Universal Robots PolyScope program: vino 4binf.urp

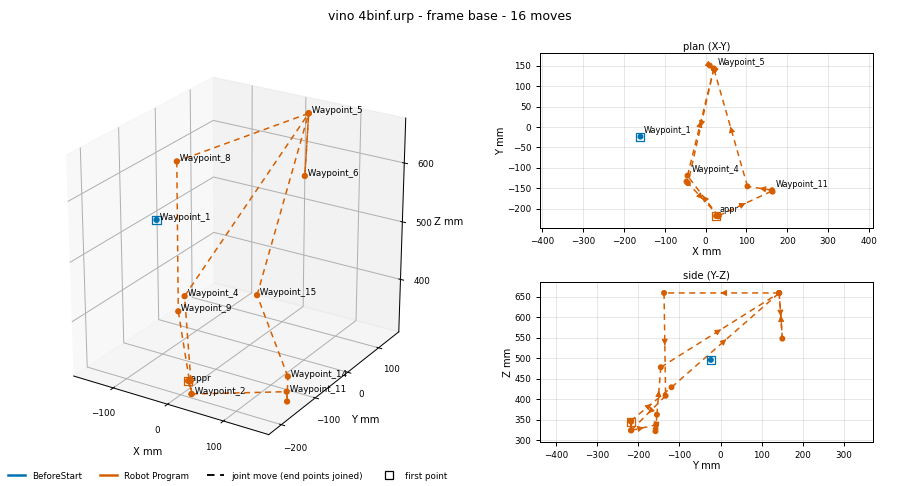
[picture p0: tool path of vino 4binf.urp in frame base, 16 of 16 moves have a stored position in this frame; points joined in program order, loops and branches not executed]
Program vino 4binf (installation=default directory=/programs createdIn=3.15.8.106339 lastSavedIn=3.15.8.106339 robotSerialNumber=2023330215)
Calibrated DH parameters: a=[-0.000158, -0.243568, -0.211872, 0.000029, -0.000046, 0]; d=[0.151957, 0.552568, 8.396945, -8.837237, 0.085345, 0.082393]; alpha=[1.571201, -0.003022, 0.002719, 1.570411, -1.571935, 0]; deltaTheta=[0.000034, -0.006936, 0.121129, -0.114397, -0.000018, 0.00002]
BeforeStart
  MoveJ speed 60 deg/s, acceleration 80 deg/s^2 (useActiveTCP=true)
    Waypoint Waypoint_1: TCP in base x=-159.567 y=-23.557 z=496.076 mm, rx=0.0292 ry=0.0156 rz=0.8759 rad; joints [-35.648, -8.811, -153.056, 70.106, 89.674, 175.859] deg; flange x=-163.543 y=-20.575 z=341.155 mm, rx=0.0292 ry=0.0156 rz=0.8759 rad
    URCap SG Grip (OnRobot, OnRobot A/S) dataModel(sg-target-width-percent=86.0)
Robot Program (runOnlyOnce=false)
  var_1 :=  (valueSource=Operator message=vino rosso:1, vino bianco:2 valueType=Integer)
  If var_1==1
    MoveJ speed 60 deg/s, acceleration 80 deg/s^2 (useActiveTCP=true)
      Waypoint appr: TCP in base x=25.587 y=-217.557 z=345.361 mm, rx=2.1967 ry=1.4969 rz=-0.0064 rad; joints [-47.133, -54.408, -74.542, -113.583, 85.897, 153.346] deg; flange x=-14.398 y=-157.633 z=482.603 mm, rx=2.1967 ry=1.4969 rz=-0.0064 rad
      Waypoint Waypoint_2: TCP in base x=31.419 y=-217.434 z=324.644 mm, rx=2.246 ry=1.4994 rz=0.0175 rad; joints [-47.147, -53.734, -79.907, -111.195, 86.968, 154.753] deg; flange x=-6.909 y=-163.472 z=464.801 mm, rx=2.246 ry=1.4994 rz=0.0175 rad
      URCap SG Grip (OnRobot, OnRobot A/S) dataModel(sg-target-width-percent=20.0, payload-weight=2.0)
      Waypoint Waypoint_3: TCP in base x=31.206 y=-218.665 z=347.338 mm, rx=2.2913 ry=1.5328 rz=-0.0001 rad; joints [-47.151, -61.647, -65.94, -120.54, 86.724, 154.677] deg; flange x=-1.134 y=-170.293 z=491.002 mm, rx=2.2913 ry=1.5328 rz=-0.0001 rad
      Waypoint Waypoint_4: TCP in base x=-44.405 y=-119.172 z=429.403 mm, rx=1.9047 ry=1.2932 rz=0.1456 rad; joints [-47.179, -40.473, -51.871, -129.238, 89.687, 154.311] deg; flange x=-122.306 y=-33.483 z=532.426 mm, rx=1.9047 ry=1.2932 rz=0.1456 rad
      MoveJ speed 60 deg/s, acceleration 80 deg/s^2 (useActiveTCP=true)
        Waypoint Waypoint_5: TCP in base x=20.05 y=142.744 z=658.935 mm, rx=1.2454 ry=-1.634 rz=-1.9818 rad; joints [-217.962, -70.658, 4.281, -114.39, 87.004, 154.418] deg; flange x=137.145 y=41.214 z=661.225 mm, rx=1.2454 ry=-1.634 rz=-1.9818 rad
        Wait Sleep waitTime=2
        Waypoint Waypoint_6: TCP in base x=9.998 y=150.468 z=547.731 mm, rx=1.5437 ry=-1.9858 rz=-1.5274 rad; joints [-217.959, -70.753, 4.268, -140.009, 87.003, 154.445] deg; flange x=114.246 y=59.022 z=616.978 mm, rx=1.5437 ry=-1.9858 rz=-1.5274 rad
        Wait Sleep waitTime=1
        Waypoint Waypoint_7: TCP in base x=20.075 y=142.736 z=658.923 mm, rx=1.2454 ry=-1.634 rz=-1.9819 rad; joints [-217.962, -70.654, 4.28, -114.394, 87.002, 154.414] deg; flange x=137.166 y=41.2 z=661.214 mm, rx=1.2454 ry=-1.634 rz=-1.9819 rad
        MoveJ speed 60 deg/s, acceleration 80 deg/s^2 (useActiveTCP=true)
          Waypoint Waypoint_8: TCP in base x=-43.492 y=-137.422 z=658.955 mm, rx=1.3394 ry=0.8543 rz=0.1901 rad; joints [-47.527, -70.659, 4.283, -114.386, 87.005, 154.417] deg; flange x=-142.09 y=-17.846 z=661.232 mm, rx=1.3394 ry=0.8543 rz=0.1901 rad
          Waypoint Waypoint_9: TCP in base x=-46.796 y=-133.623 z=408.73 mm, rx=1.9227 ry=1.2652 rz=0.0928 rad; joints [-47.145, -35.139, -63.529, -123.112, 86.887, 154.749] deg; flange x=-118.779 y=-43.172 z=511.988 mm, rx=1.9227 ry=1.2652 rz=0.0928 rad
          Waypoint Waypoint_10: TCP in base x=31.441 y=-217.42 z=324.618 mm, rx=2.246 ry=1.4996 rz=0.0176 rad; joints [-47.142, -53.734, -79.911, -111.196, 86.97, 154.751] deg; flange x=-6.888 y=-163.473 z=464.781 mm, rx=2.246 ry=1.4996 rz=0.0176 rad
          URCap SG Release (OnRobot, OnRobot A/S) dataModel(sg-target-width-percent=80.0)
  ElseIf var_1==2
    MoveJ speed 60 deg/s, acceleration 80 deg/s^2 (useActiveTCP=true)
      Waypoint Waypoint_11: TCP in base x=161.964 y=-156.646 z=337.88 mm, rx=1.2717 ry=2.6052 rz=-0.07 rad; joints [-4.628, -69.227, -57.746, -130.989, 82.548, 136.638] deg; flange x=131.859 y=-133.75 z=488.195 mm, rx=1.2717 ry=2.6052 rz=-0.07 rad
      Waypoint Waypoint_12: TCP in base x=163.817 y=-158.291 z=322.529 mm, rx=1.2225 ry=2.715 rz=-0.1341 rad; joints [-4.626, -71.776, -58.858, -132.284, 82.187, 133.389] deg; flange x=146.869 y=-135.476 z=474.901 mm, rx=1.2225 ry=2.715 rz=-0.1341 rad
      URCap SG Grip (OnRobot, OnRobot A/S) dataModel(sg-target-width-percent=20.0, payload-weight=2.0)
      Waypoint Waypoint_14: TCP in base x=162.61 y=-154.735 z=362.751 mm, rx=1.1873 ry=2.6322 rz=-0.0596 rad; joints [-4.664, -74.508, -44.621, -137.843, 83.046, 133.105] deg; flange x=129.784 y=-133.028 z=512.672 mm, rx=1.1873 ry=2.6322 rz=-0.0596 rad
      Waypoint Waypoint_15: TCP in base x=102.371 y=-145.268 z=478.205 mm, rx=0.9333 ry=2.1967 rz=0.1637 rad; joints [-4.666, -69.063, -14.745, -142.821, 84.155, 129.036] deg; flange x=-1.732 y=-120.947 z=590.438 mm, rx=0.9333 ry=2.1967 rz=0.1637 rad
      Waypoint Waypoint_16: TCP in base x=20.042 y=142.769 z=658.926 mm, rx=1.2454 ry=-1.6341 rz=-1.9818 rad; joints [-217.96, -70.659, 4.28, -114.392, 87, 154.419] deg; flange x=137.133 y=41.234 z=661.225 mm, rx=1.2454 ry=-1.6341 rz=-1.9818 rad
